DATA_BLOCK "DB_FixReadReal"
{ S7_Optimized_Access := 'FALSE' }
VERSION : 0.0
   STRUCT
      R0 : Real;
      R4 : Real;
      R8 : Real;
      R12 : Real;
      R16 : Real;
      R20 : Real;
      R24 : Real;
      R28 : Real;
      R32 : Real;
      R36 : Real;
      R40 : Real;
      R44 : Real;
      R48 : Real;
      R52 : Real;
      R56 : Real;
      R60 : Real;   // M501.M2 BQ2 actual position mm MLD (zone 1 big wheels part)
      R64 : Real;   // M501.M3 BQ3 actual position mm MLD (zone 2 big wheels part)
      R68 : Real;
      R72 : Real;
      R76 : Real;
      R80 : Real;
      R84 : Real;
      R88 : Real;
      R92 : Real;
      R96 : Real;
      R100 : Real;
      R104 : Real;
      R108 : Real;
      R112 : Real;
      R116 : Real;
      R120 : Real;   // M502.M1 BQ1actual position mm
      R124 : Real;
      R128 : Real;
      R132 : Real;
      R136 : Real;
      R140 : Real;
      R144 : Real;
      R148 : Real;
      R152 : Real;
      R156 : Real;
      R160 : Real;
      R164 : Real;
      R168 : Real;
      R172 : Real;
      R176 : Real;
      R180 : Real;   // M503
      R184 : Real;
      R188 : Real;
      R192 : Real;
      R196 : Real;
      R200 : Real;
      R204 : Real;
      R208 : Real;
      R212 : Real;
      R216 : Real;
      R220 : Real;
      R224 : Real;
      R228 : Real;
      R232 : Real;
      R236 : Real;
      R240 : Real;   // M504
      R244 : Real;
      R248 : Real;
      R252 : Real;
      R256 : Real;
      R260 : Real;
      R264 : Real;
      R268 : Real;
      R272 : Real;
      R276 : Real;
      R280 : Real;
      R284 : Real;
      R288 : Real;
      R292 : Real;
      R296 : Real;
      R300 : Real;   // M505
      R304 : Real;
      R308 : Real;
      R312 : Real;
      R316 : Real;
      R320 : Real;
      R324 : Real;
      R328 : Real;
      R332 : Real;
      R336 : Real;
      R340 : Real;
      R344 : Real;
      R348 : Real;
      R352 : Real;
      R356 : Real;
      R360 : Real;   // M506.M1(left part) BQ1actual position (flow dir.)mm
      R364 : Real;   // M506.M2 (right part) BQ2actual position (flow dir.) mm
      R368 : Real;   // M506 BQ3 (left part lateral) encoder position (mm)
      R372 : Real;   // M506 BQ4 (right part lateral) encoder position (mm)
      R376 : Real;
      R380 : Real;
      R384 : Real;
      R388 : Real;
      R392 : Real;
      R396 : Real;
      R400 : Real;
      R404 : Real;
      R408 : Real;
      R412 : Real;
      R416 : Real;
      R420 : Real;
      R424 : Real;
      R428 : Real;
      R432 : Real;
      R436 : Real;
      R440 : Real;
      R444 : Real;
      R448 : Real;
      R452 : Real;
      R456 : Real;
      R460 : Real;
      R464 : Real;
      R468 : Real;
      R472 : Real;
      R476 : Real;
      R480 : Real;
      R484 : Real;
      R488 : Real;
      R492 : Real;
      R496 : Real;
   END_STRUCT;


BEGIN
   R104 := 6.0;
   R128 := 149.5241;
   R192 := -66.20112;
   R200 := -76.06335;
   R300 := -4029.408;
   R316 := 3331.177;
   R320 := -138.2032;
   R364 := 1.45126E-38;
   R368 := 1984.16;
   R372 := 1140.075;
   R400 := -4.943526;
   R440 := -34.01926;
   R448 := -33.99865;

END_DATA_BLOCK

DATA_BLOCK "DB_FixReadDint"
{ S7_Optimized_Access := 'FALSE' }
VERSION : 0.0
   STRUCT
      DW0 : DInt;   // General.
      DW4 : DInt;
      DW8 : DInt;
      DW12 : DInt;
      DW16 : DInt;
      DW20 : DInt;
      DW24 : DInt;
      DW28 : DInt;
      DW32 : DInt;
      DW36 : DInt;
      DW40 : DInt;
      DW44 : DInt;
      DW48 : DInt;
      DW52 : DInt;
      DW56 : DInt;
      DW60 : DInt;   // M501
      DW64 : DInt;
      DW68 : DInt;
      DW72 : DInt;
      DW76 : DInt;
      DW80 : DInt;
      DW84 : DInt;
      DW88 : DInt;
      DW92 : DInt;
      DW96 : DInt;
      DW100 : DInt;
      DW104 : DInt;
      DW108 : DInt;
      DW112 : DInt;
      DW116 : DInt;
      DW120 : DInt;   // M502
      DW124 : DInt;
      DW128 : DInt;
      DW132 : DInt;
      DW136 : DInt;
      DW140 : DInt;
      DW144 : DInt;
      DW148 : DInt;
      DW152 : DInt;
      DW156 : DInt;
      DW160 : DInt;
      DW164 : DInt;
      DW168 : DInt;
      DW172 : DInt;
      DW176 : DInt;
      DW180 : DInt;   // M503 BQ1 Rotator encoder pulses (reading referenced to starting value)
      DW184 : DInt;
      DW188 : DInt;
      DW192 : DInt;
      DW196 : DInt;
      DW200 : DInt;
      DW204 : DInt;
      DW208 : DInt;
      DW212 : DInt;
      DW216 : DInt;
      DW220 : DInt;
      DW224 : DInt;
      DW228 : DInt;
      DW232 : DInt;
      DW236 : DInt;
      DW240 : DInt;   // M504
      DW244 : DInt;
      DW248 : DInt;
      DW252 : DInt;
      DW256 : DInt;
      DW260 : DInt;
      DW264 : DInt;
      DW268 : DInt;
      DW272 : DInt;
      DW276 : DInt;
      DW280 : DInt;
      DW284 : DInt;
      DW288 : DInt;
      DW292 : DInt;
      DW296 : DInt;
      DW300 : DInt;   // M505
      DW304 : DInt;
      DW308 : DInt;
      DW312 : DInt;
      DW316 : DInt;
      DW320 : DInt;
      DW324 : DInt;
      DW328 : DInt;
      DW332 : DInt;
      DW336 : DInt;
      DW340 : DInt;
      DW344 : DInt;
      DW348 : DInt;
      DW352 : DInt;
      DW356 : DInt;
      DW360 : DInt;   // M506
      DW364 : DInt;   // M506
      DW368 : DInt;   // M506 BQ3 (left part MLD) encoder pulses
      DW372 : DInt;   // M506 BQ4 (right part MLD) encoder pulses
      DW376 : DInt;
      DW380 : DInt;
      DW384 : DInt;
      DW388 : DInt;
      DW392 : DInt;
      DW396 : DInt;
      DW400 : DInt;
      DW404 : DInt;
      DW408 : DInt;
      DW412 : DInt;
      DW416 : DInt;
      DW420 : DInt;
      DW424 : DInt;
      DW428 : DInt;
      DW432 : DInt;
      DW436 : DInt;
      DW440 : DInt;
      DW444 : DInt;
      DW448 : DInt;
      DW452 : DInt;
      DW456 : DInt;
      DW460 : DInt;
      DW464 : DInt;
      DW468 : DInt;
      DW472 : DInt;
      DW476 : DInt;
      DW480 : DInt;   // LES1_M507:BQ1.Encoder position (imp)
      DW484 : DInt;
      DW488 : DInt;
      DW492 : DInt;
      DW496 : DInt;
      DW500 : DInt;
      DW504 : DInt;
      DW508 : DInt;
      DW512 : DInt;
      DW516 : DInt;
      DW520 : DInt;   // LES1_M508:Slide 1.BQ1.Encoder position (imp)
      DW524 : DInt;   // LES1_M508:Slide 2.BQ2.Encoder position (imp)
      DW528 : DInt;   // LES1_M508:Slide 1.BQ1.Encoder position (mm)
      DW532 : DInt;   // LES1_M508:Slide 2.BQ2.Encoder position (mm)
      DW536 : DInt;
      DW540 : DInt;
      DW544 : DInt;
      DW548 : DInt;
      DW552 : DInt;
      DW556 : DInt;
      DW560 : DInt;
      DW564 : DInt;
      DW568 : DInt;
      DW572 : DInt;
      DW576 : DInt;
      DW580 : DInt;
      DW584 : DInt;   // LES1_M508:Rotating platform.BQ3.Encoder position (imp)
      DW588 : DInt;
      DW592 : DInt;
      DW596 : DInt;
      DW600 : DInt;
      DW604 : DInt;
      DW608 : DInt;
      DW612 : DInt;
      DW616 : DInt;
      DW620 : DInt;
      DW624 : DInt;
      DW628 : DInt;
      DW632 : DInt;
      DW636 : DInt;
      DW640 : DInt;
      DW644 : DInt;
      DW648 : DInt;
      DW652 : DInt;
      DW656 : DInt;
      DW660 : DInt;
      DW664 : DInt;
      DW668 : DInt;
      DW672 : DInt;
      DW676 : DInt;
      DW680 : DInt;
      DW684 : DInt;
      DW688 : DInt;
      DW692 : DInt;
      DW696 : DInt;
      DW700 : DInt;
      DW704 : DInt;
      DW708 : DInt;
      DW712 : DInt;
      DW716 : DInt;
      DW720 : DInt;
      DW724 : DInt;
      DW728 : DInt;
      DW732 : DInt;
      DW736 : DInt;
      DW740 : DInt;
      DW744 : DInt;
      DW748 : DInt;
      DW752 : DInt;
      DW756 : DInt;
      DW760 : DInt;
      DW764 : DInt;
      DW768 : DInt;
      DW772 : DInt;
      DW776 : DInt;
      DW780 : DInt;
      DW784 : DInt;
      DW788 : DInt;
      DW792 : DInt;
      DW796 : DInt;
      DW800 : DInt;
      DW804 : DInt;
      DW808 : DInt;
      DW812 : DInt;
      DW816 : DInt;
      DW820 : DInt;
      DW824 : DInt;
      DW828 : DInt;
      DW832 : DInt;
      DW836 : DInt;
      DW840 : DInt;
      DW844 : DInt;
      DW848 : DInt;
      DW852 : DInt;
      DW856 : DInt;
      DW860 : DInt;
      DW864 : DInt;
      DW868 : DInt;
      DW872 : DInt;
      DW876 : DInt;
      DW880 : DInt;
      DW884 : DInt;
      DW888 : DInt;
      DW892 : DInt;
      DW896 : DInt;
   END_STRUCT;


BEGIN
   DW128 := DINT#14373;
   DW368 := DINT#79289;
   DW372 := DINT#27030;
   DW384 := DINT#2300;
   DW392 := DINT#4600;
   DW404 := DINT#3210;
   DW432 := DINT#1605;
   DW480 := DINT#1363;
   DW520 := DINT#7471;
   DW524 := DINT#7728;
   DW528 := DINT#912;
   DW532 := DINT#943;
   DW536 := DINT#91114;
   DW584 := DINT#27181;

END_DATA_BLOCK

DATA_BLOCK "DB_FixReadInt"
{ S7_Optimized_Access := 'FALSE' }
VERSION : 0.0
   STRUCT
      W0 : Int;   // Z500. State zone
      W2 : Int;
      W4 : Int;   // Z500.Mode zone (1=manu  4=auto)
      W6 : Int;
      W8 : Int;
      W10 : Int;   // Z500.selected (1=20;3=40 4=60 5=80 m/min)
      W12 : Int;
      W14 : Int;   // Z500 anomaly on  MCC1501 (1=faute)
      W16 : Int;
      W18 : Int;   // Z500. Line Enable (1=enable 0=no )
      W20 : Int;   // Z500. Line ready to receive glass from Main line (1= ready  0= Not ready)
      W22 : Int;
      W24 : Int;   // Z500.Selection conveyor start clean (M501-M506)(accepted)
      W26 : Int;
      W28 : Int;
      BitNuovi : Struct   // struct created to use this word, relative to "Portrait=1 /Landscape=2" as a bit
         byteMSD : Byte;
         bit0 : Bool;   // Z500.selected Unloading mode =Portrait
         bit1 : Bool;   // Z500.Selected Unloading mode =Landscape
      END_STRUCT;
      W32 : Int;
      W34 : Int;
      W36 : Int;
      W38 : Int;
      W40 : Int;
      W42 : Int;
      W44 : Int;
      W46 : Int;
      W48 : Int;
      W50 : Int;   // M501.M1.Machine state (rollers part)
      W52 : Int;   // M501.M2.Machine state (zone 1 wheels part)
      W54 : Int;   // M501.M3.Machine state (zone 2 wheels part)
      W56 : Int;   // M501.M4.Machine state (glass unload)
      W58 : Int;
      W60 : Int;
      W62 : Int;
      W64 : Int;
      W66 : Int;
      W68 : Int;
      W70 : Int;   // M502.M1.Machine state
      W72 : Int;   // M502_3 Area access status
      W74 : Int;
      W76 : Int;
      W78 : Int;
      W80 : Int;
      W82 : Int;
      W84 : Int;
      W86 : Int;
      W88 : Int;
      W90 : Int;   // M503.Machine state (Rotator device)
      W92 : Int;
      W94 : Int;
      W96 : Int;
      W98 : Int;
      W100 : Int;
      W102 : Int;
      W104 : Int;
      W106 : Int;
      W108 : Int;
      W110 : Int;   // M504.M1 Machine state (left)
      W112 : Int;   // M504.M2 Machine state (right)
      W114 : Int;
      W116 : Int;   // M504 Speed reduction during unpacking status  (0= OFF 1= ON)
      W118 : Int;   // M504 Move Backward enable status (0= OFF 1= ON)
      W120 : Int;
      W122 : Int;
      W124 : Int;
      W126 : Int;
      W128 : Int;
      W130 : Int;   // M505.M1 Machine state (left)
      W132 : Int;   // M505.M2 Machine state (right)
      W134 : Int;
      W136 : Int;
      W138 : Int;
      W140 : Int;
      W142 : Int;
      W144 : Int;
      W146 : Int;
      W148 : Int;
      W150 : Int;   // M506.M1 Machine state (left)
      W152 : Int;   // M506.M2 Machine state (right)
      W154 : Int;   // M506.M3 Machine state (left) MLD
      W156 : Int;   // M506.M4 Machine state (right) MLD
      W158 : Int;   // M506 Right Glass Presence status (1=Loaded 2=Positione 4=Squared) A or Mono
      W160 : Int;   // M506 Left Glass Presence status (1=Loaded 2=Positione 4=Squared) B
      W162 : Int;
      W164 : Int;
      W166 : Int;
      W168 : Int;
      W170 : Int;
      W172 : Int;
      W174 : Int;
      W176 : Int;
      W178 : Int;
      W180 : Int;
      W182 : Int;
      W184 : Int;
      W186 : Int;
      W188 : Int;
      W190 : Int;
      W192 : Int;
      W194 : Int;
      W196 : Int;
      W198 : Int;
      W200 : Int;
      W202 : Int;
      W204 : Int;
      W206 : Int;
      W208 : Int;
      W210 : Int;
      W212 : Int;
      W214 : Int;
      W216 : Int;
      W218 : Int;
      W220 : Int;
      W222 : Int;
      W224 : Int;
      W226 : Int;
      W228 : Int;
      W230 : Int;   // LES1_M507.Entry Zone
      W232 : Int;   // LES1_M507.Entry Zone Barriere Photocell
      W234 : Int;   // LES1_M507.Entry Zone door
      W236 : Int;   // LES1_M507.Cycle Time (s/100)
      W238 : Int;   // LES1_M507.Test Modality (1=Active)
      W240 : Int;   // LES1_M507.Arm Speed selection (1=Selection,0=Thickness)
      W242 : Int;   // LES1_M507 Cups selection in manual(1) or auto(0)
      W244 : Int;
      W246 : Int;
      W248 : Int;
      W250 : Int;
      W252 : Int;
      W254 : Int;
      W256 : Int;
      W258 : Int;
      W260 : Int;   // LES1_M507:State machine(1,3,7)
      W262 : Int;   // LES1_M507:Mode machine(Manu,semiauto,auto) 1,2,4
      W264 : Int;   // LES1_M507.Actual arms speed
      W266 : Int;   // LES1_M507:Status return in line ( 0=NoReentry 1=ReentryReq. 2=ReentryAccepted)
      W268 : Int;
      W270 : Int;   // M507_Z.St.:1=Stop2=Starting3=Run 4=Stop 7=Fault 15=Clean line 16=Emerg. 17=Man
      W272 : Int;
      W274 : Int;
      W276 : Int;   // LES1 :M507 Actual arms position
      W278 : Int;
      W280 : Int;   // LES1_M507:glass presence (0= no glass 1= presence 1 sheet  2=presence 2 sheets)
      W282 : Int;
      W284 : Int;
      W286 : Int;
      W288 : Int;
      W290 : Int;   // LES1_M507.Legth (mm)
      W292 : Int;   // LES1_M507.Whidth (mm)
      W294 : Int;   // LES1_M507.Thickness (mm/100)
      W296 : Int;
      W298 : Int;
      W300 : Int;   // LES1_M507: (0= DISABLED  1= ENABLE)
      W302 : Int;
      W304 : Int;
      W306 : Int;
      W308 : Int;
      W310 : Int;
      W312 : Int;
      W314 : Int;
      W316 : Int;
      W318 : Int;
      W320 : Int;
      W322 : Int;
      W324 : Int;
      W326 : Int;
      W328 : Int;
      W330 : Int;
      W332 : Int;
      W334 : Int;
      W336 : Int;
      W338 : Int;
      W340 : Int;
      W342 : Int;
      W344 : Int;
      W346 : Int;
      W348 : Int;
      W350 : Int;
      W352 : Int;
      W354 : Int;
      W356 : Int;
      W358 : Int;
      W360 : Int;   // LES1_M508:State machine (plateform)
      W362 : Int;   // LES1_M508:State machine (slide 1)
      W364 : Int;   // LES1_M508:State machine (slide 2)
      W366 : Int;   // LES1_M508.Platform Data Source (0=FIX 1=Remote)
      W368 : Int;   // LES1_M508.Platform Rack State 1= aligned side A
      W370 : Int;   // LES1_M508.Platform Rack State 1= aligned side B
      W372 : Int;   // LES1_M508.Platform 0° Side A (0=Not Ready, 1=Ready)
      W374 : Int;   // LES1_M508.Platform 180° Side B (0=Not Ready, 1=Ready)
      W376 : Int;   // LES1_M508.Platform 0°  Set Pack number
      W378 : Int;   // LES1_M508.Platform 0°  Set Sheet number
      W380 : Int;   // LES1_M508.Platform 0° Unloaded Pack
      W382 : Int;   // LES1_M508.Platform 0° Unloaded Sheet
      W384 : Int;
      W386 : Int;   // LES1_M508.Platform 180°  Set Pack number
      W388 : Int;   // LES1_M508.Platform 180°  Set Sheet number
      W390 : Int;   // LES1_M508.Platform 180° Unloaded Pack
      W392 : Int;   // LES1_M508.Platform 180° Unloaded Sheet
      W394 : Int;
      W396 : Int;
      W398 : Int;
      W400 : Int;   // LES1 M508.Slides Selection cycle type (1 = Fixed, 0 = Thickness)
      W402 : Int;
      W404 : Int;
      W406 : Int;
      W408 : Int;
      W410 : Int;
      W412 : Int;
      W414 : Int;
      W416 : Int;
      W418 : Int;
      W420 : Int;
      W422 : Int;
      W424 : Int;
      W426 : Int;
      W428 : Int;
      W430 : Int;   // LES1_M509 left pusher :State machine (1,3,7)
      W432 : Int;   // LES1_M509 right pusher :State machine (1,3,7)
      W434 : Int;
      W436 : Int;
      W438 : Int;
      W440 : Int;
      W442 : Int;
      W444 : Int;
      W446 : Int;
      W448 : Int;
      W450 : Int;
      W452 : Int;
      W454 : Int;
      W456 : Int;
      W458 : Int;
      W460 : Int;
      W462 : Int;
      W464 : Int;
      W466 : Int;
      W468 : Int;
      W470 : Int;
      W472 : Int;
      W474 : Int;
      W476 : Int;
      W478 : Int;
      W480 : Int;
      W482 : Int;
      W484 : Int;
      W486 : Int;
      W488 : Int;
      W490 : Int;
      W492 : Int;
      W494 : Int;
      W496 : Int;
      W498 : Int;
      W500 : Int;
      W502 : Int;
      W504 : Int;
      W506 : Int;
      W508 : Int;
      W510 : Int;
      W512 : Int;
      W514 : Int;
      W516 : Int;
      W518 : Int;
      W520 : Int;
      W522 : Int;
      W524 : Int;
      W526 : Int;
      W528 : Int;
      W530 : Int;
      W532 : Int;
      W534 : Int;
      W536 : Int;
      W538 : Int;
      W540 : Int;
      W542 : Int;
      W544 : Int;
      W546 : Int;
      W548 : Int;
      W550 : Int;
      W552 : Int;
      W554 : Int;
      W556 : Int;
      W558 : Int;
      W560 : Int;
      W562 : Int;
      W564 : Int;
      W566 : Int;
      W568 : Int;
      W570 : Int;
      W572 : Int;
      W574 : Int;
      W576 : Int;
      W578 : Int;
      W580 : Int;
      W582 : Int;
      W584 : Int;
      W586 : Int;
      W588 : Int;
      W590 : Int;
      W592 : Int;
      W594 : Int;
      W596 : Int;
      W598 : Int;
      W600 : Int;
      W602 : Int;
      W604 : Int;
      W606 : Int;
      W608 : Int;
      W610 : Int;
      W612 : Int;
      W614 : Int;
      W616 : Int;
      W618 : Int;
      W620 : Int;
      W622 : Int;
      W624 : Int;
      W626 : Int;
      W628 : Int;
      W630 : Int;
      W632 : Int;
      W634 : Int;
      W636 : Int;
      W638 : Int;
      W640 : Int;
      W642 : Int;
      W644 : Int;
      W646 : Int;
      W648 : Int;
      W650 : Int;
      W652 : Int;
      W654 : Int;
      W656 : Int;
      W658 : Int;
      W660 : Int;
      W662 : Int;
      W664 : Int;
      W666 : Int;
      W668 : Int;
      W670 : Int;
      W672 : Int;
      W674 : Int;
      W676 : Int;
      W678 : Int;
      W680 : Int;
      W682 : Int;
      W684 : Int;
      W686 : Int;
      W688 : Int;
      W690 : Int;
      W692 : Int;
      W694 : Int;
      W696 : Int;
      W698 : Int;
      W700 : Int;
      W702 : Int;
      W704 : Int;
      W706 : Int;
      W708 : Int;
      W710 : Int;
      W712 : Int;
      W714 : Int;
      W716 : Int;
      W718 : Int;
      W720 : Int;
      W722 : Int;
      W724 : Int;
      W726 : Int;
      W728 : Int;
      W730 : Int;
      W732 : Int;
      W734 : Int;
      W736 : Int;
      W738 : Int;
      W740 : Int;
      W742 : Int;
      W744 : Int;
      W746 : Int;
      W748 : Int;
      W750 : Int;
      W752 : Int;
      W754 : Int;
      W756 : Int;
      W758 : Int;
      W760 : Int;
      W762 : Int;
      W764 : Int;
      W766 : Int;
      W768 : Int;
      W770 : Int;
      W772 : Int;
      W774 : Int;
      W776 : Int;
      W778 : Int;
      W780 : Int;
      W782 : Int;
      W784 : Int;
      W786 : Int;
      W788 : Int;
      W790 : Int;
      W792 : Int;
      W794 : Int;
      W796 : Int;
      W798 : Int;
      W800 : Int;
      W802 : Int;
      W804 : Int;
      W806 : Int;
      W808 : Int;
      W810 : Int;
      W812 : Int;
      W814 : Int;
      W816 : Int;
      W818 : Int;
      W820 : Int;
      W822 : Int;
      W824 : Int;
      W826 : Int;
      W828 : Int;
      W830 : Int;
      W832 : Int;
      W834 : Int;
      W836 : Int;
      W838 : Int;
      W840 : Int;
      W842 : Int;
      W844 : Int;
      W846 : Int;
      W848 : Int;
      W850 : Int;
      W852 : Int;
      W854 : Int;
      W856 : Int;
      W858 : Int;
      W860 : Int;
      W862 : Int;
      W864 : Int;
      W866 : Int;
      W868 : Int;
      W870 : Int;
      W872 : Int;
      W874 : Int;
      W876 : Int;
      W878 : Int;
      W880 : Int;
      W882 : Int;
      W884 : Int;
      W886 : Int;
      W888 : Int;
      W890 : Int;
      W892 : Int;
      W894 : Int;
      W896 : Int;
      W898 : Int;
      W900 : Int;
      W902 : Int;
      W904 : Int;
      W906 : Int;
      W908 : Int;
      W910 : Int;
      W912 : Int;
      W914 : Int;
      W916 : Int;
      W918 : Int;
      W920 : Int;
      W922 : Int;
      W924 : Int;
      W926 : Int;
      W928 : Int;
      W930 : Int;
      W932 : Int;
      W934 : Int;
      W936 : Int;
      W938 : Int;
      W940 : Int;
      W942 : Int;
      W944 : Int;
      W946 : Int;
      W948 : Int;
      W950 : Int;
      W952 : Int;
      W954 : Int;
      W956 : Int;
      W958 : Int;
      W960 : Int;
      W962 : Int;
      W964 : Int;
      W966 : Int;
      W968 : Int;
      W970 : Int;
      W972 : Int;
      W974 : Int;
      W976 : Int;
      W978 : Int;
      W980 : Int;
      W982 : Int;
      W984 : Int;
      W986 : Int;
      W988 : Int;
      W990 : Int;
      W992 : Int;
      W994 : Int;
      W996 : Int;
      W998 : Int;
      W1000 : Int;
      W1002 : Int;
      W1004 : Int;
      W1006 : Int;
      W1008 : Int;
      W1010 : Int;
      W1012 : Int;
      W1014 : Int;
      W1016 : Int;
      W1018 : Int;
      W1020 : Int;
      W1022 : Int;
      W1024 : Int;
      W1026 : Int;
      W1028 : Int;
      W1030 : Int;
      W1032 : Int;
      W1034 : Int;
      W1036 : Int;
      W1038 : Int;
      W1040 : Int;
      W1042 : Int;
      W1044 : Int;
      W1046 : Int;
      W1048 : Int;
      W1050 : Int;
      W1052 : Int;
      W1054 : Int;
      W1056 : Int;
      W1058 : Int;
      W1060 : Int;
      W1062 : Int;
      W1064 : Int;
      W1066 : Int;
      W1068 : Int;
      W1070 : Int;
      W1072 : Int;
      W1074 : Int;
      W1076 : Int;
      W1078 : Int;
      W1080 : Int;
      W1082 : Int;
      W1084 : Int;
      W1086 : Int;
      W1088 : Int;
      W1090 : Int;
      W1092 : Int;
      W1094 : Int;
      W1096 : Int;
      W1098 : Int;
      W1100 : Int;
      W1102 : Int;
      W1104 : Int;
      W1106 : Int;
      W1108 : Int;
      W1110 : Int;
      W1112 : Int;
      W1114 : Int;
      W1116 : Int;
      W1118 : Int;
      W1120 : Int;
      W1122 : Int;
      W1124 : Int;
      W1126 : Int;
      W1128 : Int;
      W1130 : Int;
      W1132 : Int;
      W1134 : Int;
      W1136 : Int;
      W1138 : Int;
      W1140 : Int;
      W1142 : Int;
      W1144 : Int;
      W1146 : Int;
      W1148 : Int;
      W1150 : Int;
      W1152 : Int;
      W1154 : Int;
      W1156 : Int;
      W1158 : Int;
      W1160 : Int;
      W1162 : Int;
      W1164 : Int;
      W1166 : Int;
      W1168 : Int;
      W1170 : Int;
      W1172 : Int;
      W1174 : Int;
      W1176 : Int;
      W1178 : Int;
      W1180 : Int;
      W1182 : Int;
      W1184 : Int;
      W1186 : Int;
      W1188 : Int;
      W1190 : Int;
      W1192 : Int;
      W1194 : Int;
      W1196 : Int;
      W1198 : Int;
      W1200 : Int;
      W1202 : Int;
      W1204 : Int;
      W1206 : Int;
      W1208 : Int;
      W1210 : Int;
      W1212 : Int;
      W1214 : Int;
      W1216 : Int;
      W1218 : Int;
      W1220 : Int;
      W1222 : Int;
      W1224 : Int;
      W1226 : Int;
      W1228 : Int;
      W1230 : Int;
      W1232 : Int;
      W1234 : Int;
      W1236 : Int;
      W1238 : Int;
      W1240 : Int;
      W1242 : Int;
      W1244 : Int;
      W1246 : Int;
      W1248 : Int;
      W1250 : Int;
      W1252 : Int;
      W1254 : Int;
      W1256 : Int;
      W1258 : Int;
      W1260 : Int;
      W1262 : Int;
      W1264 : Int;
      W1266 : Int;
      W1268 : Int;
      W1270 : Int;
      W1272 : Int;
      W1274 : Int;
      W1276 : Int;
      W1278 : Int;
      W1280 : Int;
      W1282 : Int;
      W1284 : Int;
      W1286 : Int;
      W1288 : Int;
      W1290 : Int;
      W1292 : Int;
      W1294 : Int;
      W1296 : Int;
      W1298 : Int;
      W1300 : Int;
      W1302 : Int;
      W1304 : Int;
      W1306 : Int;
      W1308 : Int;
      W1310 : Int;
      W1312 : Int;
      W1314 : Int;
      W1316 : Int;
      W1318 : Int;
      W1320 : Int;
      W1322 : Int;
      W1324 : Int;
      W1326 : Int;
      W1328 : Int;
      W1330 : Int;
      W1332 : Int;
      W1334 : Int;
      W1336 : Int;
      W1338 : Int;
      W1340 : Int;
      W1342 : Int;
      W1344 : Int;
      W1346 : Int;
      W1348 : Int;
      W1350 : Int;
      W1352 : Int;
      W1354 : Int;
      W1356 : Int;
      W1358 : Int;
      W1360 : Int;
      W1362 : Int;
      W1364 : Int;
      W1366 : Int;
      W1368 : Int;
      W1370 : Int;
      W1372 : Int;
      W1374 : Int;
      W1376 : Int;
      W1378 : Int;
      W1380 : Int;
      W1382 : Int;
      W1384 : Int;
      W1386 : Int;
      W1388 : Int;
      W1390 : Int;
      W1392 : Int;
      W1394 : Int;
      W1396 : Int;
      W1398 : Int;
      W1400 : Int;
      W1402 : Int;
      W1404 : Int;
      W1406 : Int;
      W1408 : Int;
      W1410 : Int;
      W1412 : Int;
      W1414 : Int;
      W1416 : Int;
      W1418 : Int;
      W1420 : Int;
      W1422 : Int;
      W1424 : Int;
      W1426 : Int;
      W1428 : Int;
      W1430 : Int;
      W1432 : Int;
      W1434 : Int;
      W1436 : Int;
      W1438 : Int;
      W1440 : Int;
      W1442 : Int;
      W1444 : Int;
      W1446 : Int;
      W1448 : Int;
      W1450 : Int;
      W1452 : Int;
      W1454 : Int;
      W1456 : Int;
      W1458 : Int;
      W1460 : Int;
      W1462 : Int;
      W1464 : Int;
      W1466 : Int;
      W1468 : Int;
      W1470 : Int;
      W1472 : Int;
      W1474 : Int;
      W1476 : Int;
      W1478 : Int;
      W1480 : Int;
      W1482 : Int;
      W1484 : Int;
      W1486 : Int;
      W1488 : Int;
      W1490 : Int;
      W1492 : Int;
      W1494 : Int;
      W1496 : Int;
      W1498 : Int;
   END_STRUCT;


BEGIN
   W0 := 3;
   W4 := 4;
   W10 := 4;
   W18 := 1;
   W20 := 1;
   W24 := 506;
   W26 := 505;
   BitNuovi.bit1 := TRUE;
   W50 := 3;
   W52 := 3;
   W54 := 3;
   W56 := 1;
   W60 := 1;
   W62 := 1;
   W64 := 1;
   W66 := 1;
   W68 := 1;
   W70 := 3;
   W74 := 7;
   W76 := 7;
   W78 := 7;
   W80 := 1;
   W82 := 1;
   W84 := 1;
   W86 := 1;
   W90 := 1;
   W92 := 7;
   W100 := 7;
   W110 := 3;
   W112 := 3;
   W118 := 1;
   W130 := 3;
   W132 := 3;
   W146 := 7;
   W150 := 3;
   W152 := 3;
   W154 := 1;
   W156 := 1;
   W166 := 1;
   W170 := 1;
   W172 := 1;
   W174 := 1;
   W178 := 1;
   W190 := 7;
   W192 := 7;
   W210 := 7;
   W218 := 1;
   W220 := 1;
   W230 := 2;
   W232 := 7;
   W234 := 1;
   W240 := 1;
   W250 := 7;
   W252 := 7;
   W258 := 1;
   W260 := 1;
   W262 := 4;
   W264 := 50;
   W270 := 3;
   W276 := 2;
   W278 := 1;
   W290 := 1830;
   W292 := 2440;
   W294 := 500;
   W298 := 1;
   W300 := 2;
   W308 := 1;
   W318 := 1;
   W338 := 1;
   W358 := 1;
   W360 := 7;
   W362 := 7;
   W364 := 1;
   W366 := 1;
   W370 := 1;
   W372 := 1;
   W374 := 1;
   W376 := 1;
   W378 := 45;
   W386 := 1;
   W388 := 45;
   W392 := 4;
   W398 := 7;
   W402 := 16;
   W404 := 3;
   W406 := 1;
   W408 := 1;
   W418 := 7;
   W422 := 7;
   W424 := 75;
   W430 := 1;
   W432 := 1;
   W436 := 6;
   W438 := 7;
   W440 := 1060;
   W442 := 1530;
   W444 := 210;
   W450 := 7;
   W452 := 1;
   W458 := 41;
   W460 := 1;
   W464 := 1;
   W466 := 252;
   W478 := 7;
   W480 := 1;
   W484 := 1;
   W486 := 252;
   W492 := 44;
   W498 := 7;
   W500 := 1;
   W510 := 7;
   W518 := 7;
   W520 := 7;
   W538 := 7;
   W550 := 1;
   W556 := 3;
   W558 := 7;
   W578 := 7;
   W596 := 1;
   W598 := 1;
   W638 := 1;
   W658 := 1;
   W678 := 1;
   W698 := 1;
   W738 := 7;
   W758 := 1;
   W778 := 20;
   W838 := 7;
   W858 := 7;
   W900 := 17;
   W914 := 1;
   W938 := 1;
   W958 := 7;
   W978 := 1;
   W998 := 1;
   W1018 := 1;
   W1038 := 1;
   W1058 := 1;
   W1078 := 1;
   W1098 := 1;
   W1118 := 7;
   W1138 := 7;
   W1158 := 7;
   W1236 := 1;
   W1238 := 1;
   W1240 := 1;
   W1242 := 1;
   W1276 := 1;
   W1278 := 1;
   W1280 := 1;
   W1282 := 1;
   W1320 := 17;
   W1322 := 1;
   W1324 := 3;
   W1358 := 7;
   W1398 := 7;

END_DATA_BLOCK

DATA_BLOCK "DB_FixReadBit"
{ S7_Optimized_Access := 'FALSE' }
VERSION : 0.0
   STRUCT
      b00 : Bool;   // A 32.0 oZ500-MCC1302-Lateral line enabled
      b01 : Bool;   // A 32.1 oZ500-MCC1302- Ready for Cap of lengh <=1830 mm
      b02 : Bool;   // A 32.2 oZ500-MCC1302-Ready for Cap of length > 1830 mm
      b03 : Bool;   // A 32.3 oZ500-MCC1302-Glass clearing lamp for M319
      b04 : Bool;   // A 32.4 oZ500-MCC1302-Unloading >> M319 in progress
      b05 : Bool;
      b06 : Bool;
      b07 : Bool;
      b10 : Bool;   // E      18.0 iZ500-MCC1302-Syncronisation by line -cap arriving
      b11 : Bool;   // E      18.1 iZ500-MCC1302-No convoy request by line
      b12 : Bool;   // E      18.2 iZ500-MCC1302-Speed by line bit 0
      b13 : Bool;   // E      18.3 iZ500-MCC1302-Speed by line bit 1
      b14 : Bool;   // E      18.4 iZ500-MCC1302-glass on tilting machine < in length of "2000 mm"
      b15 : Bool;   // E      18.5 iZ500-MCC1302-glass call clearing p.b.:M319SB4
      b16 : Bool;   // E      18.6 iZ500-MCC1302-Request disable consents by arriving SQC plate
      b17 : Bool;
      b20 : Bool;
      b21 : Bool;
      b22 : Bool;   // Z500.Force mono mode (0=not actived 1=actived)
      b23 : Bool;
      b24 : Bool;
      b25 : Bool;
      b26 : Bool;
      b27 : Bool;
      b30 : Bool;
      b31 : Bool;
      b32 : Bool;
      b33 : Bool;
      b34 : Bool;
      b35 : Bool;
      b36 : Bool;
      b37 : Bool;
      b40 : Bool;   // M501. P142KA1 photocell for positioning on M2/M3  (Start count)E67.2
      b41 : Bool;   // M501-B2 photocell of glass stop for SQC E4.0
      b42 : Bool;   // M501-B3 photocell of unpacking right side E4.1 (not really present)
      b43 : Bool;   // M501-B4 photocell of unpacking left side E4.2 (not really present)
      b44 : Bool;
      b45 : Bool;
      b46 : Bool;
      b47 : Bool;
      b50 : Bool;   // M501.P145KA1small wheels frame to high position E67.7
      b51 : Bool;
      b52 : Bool;
      b53 : Bool;
      b54 : Bool;
      b55 : Bool;
      b56 : Bool;
      b57 : Bool;
      b60 : Bool;   // M502-B1-B2 P146KA1 photocell for positioning during load E68.3
      b61 : Bool;
      b62 : Bool;
      b63 : Bool;
      b64 : Bool;
      b65 : Bool;
      b66 : Bool;
      b67 : Bool;
      b70 : Bool;
      b71 : Bool;
      b72 : Bool;
      b73 : Bool;
      b74 : Bool;
      b75 : Bool;
      b76 : Bool;
      b77 : Bool;
      b80 : Bool;   // M503 P148KA1 Frame to high position E69.0
      b81 : Bool;   // M503 P148KA2 Frame to low position E69.1
      b82 : Bool;   // M503-SQ1 Centering device confirm position E4.3
      b83 : Bool;   // M503-SQ4 Centering device opened (rot.allowed)E4.4
      b84 : Bool;   // M503-SQ5 Centering device closed (rot.not allowed)E4.5
      b85 : Bool;
      b86 : Bool;
      b87 : Bool;   // M503 request of rotation (1= request of rotation 0= no request of rotation)
      b90 : Bool;   // M503 glass rotated (1= rotated 0= not rotated)
      b91 : Bool;
      b92 : Bool;
      b93 : Bool;   // M502-M503 (area saferies)
      b94 : Bool;
      b95 : Bool;
      b96 : Bool;
      b97 : Bool;
      b100 : Bool;   // M504-B1 Glass sheet stop left transport E5.6
      b101 : Bool;   // M504-B2 Glass sheet stop right transport E5.7
      b102 : Bool;   // M504-B3 Glass sheet syncronisation left transport E7.4
      b103 : Bool;   // M504-B4 Glass sheet syncronisation right transport E7.5
      b104 : Bool;
      b105 : Bool;
      b106 : Bool;
      b107 : Bool;
      b110 : Bool;
      b111 : Bool;
      b112 : Bool;
      b113 : Bool;
      b114 : Bool;
      b115 : Bool;
      b116 : Bool;
      b117 : Bool;
      b120 : Bool;   // M505-B3 P173KA1 Glass sheet stop left E75.4
      b121 : Bool;   // M505-B4 P174KA1 Glass sheet stop right E75.6
      b122 : Bool;   // M505-B1 Glass sheet slowdown left transport E6.7
      b123 : Bool;   // M505-B2 Glass sheet slowdown right transport E7.0
      b124 : Bool;
      b125 : Bool;   // M505-SQ4 Frontal squaring upper position E7.2
      b126 : Bool;
      b127 : Bool;
      b130 : Bool;
      b131 : Bool;
      b132 : Bool;
      b133 : Bool;
      b134 : Bool;
      b135 : Bool;
      b136 : Bool;
      b137 : Bool;
      b140 : Bool;   // M506-B11 Glass sheet stop left E7.6
      b141 : Bool;   // M506-SQ11 stop backward translation left photocell E7.7
      b142 : Bool;   // M506-SQ12 stop forward translation left photocell E8.0
      b143 : Bool;   // M506-B21 Glass sheet stop right E8.1
      b144 : Bool;   // M506-SQ21 stop backward translation right photocell E8.2
      b145 : Bool;   // M506-SQ22 stop forward translation right photocell E8.3
      b146 : Bool;   // M506 -P177KA1 Frame to high position E76.4
      b147 : Bool;
      b150 : Bool;
      b151 : Bool;
      b152 : Bool;
      b153 : Bool;
      b154 : Bool;
      b155 : Bool;
      b156 : Bool;
      b157 : Bool;
      b160 : Bool;   // LES1_M507.Indexing (B1 E8.7)
      b161 : Bool;   // LES1_M507.Compressed air pressure (SP1 E9.4)
      b162 : Bool;   // LES1_M507.Change inclination backward (SQ1 E9.7)
      b163 : Bool;   // LES1_M507.Change inclination to middle (SQ2 E9.2)
      b164 : Bool;   // LES1_M507.Change inclination forward (SQ3 E9.3)
      b165 : Bool;   // LES1_M507.Preindexing (B2 E9.0)
      b166 : Bool;   // LES1_M507.Vacuum presence (SP3 E9.3)
      b167 : Bool;   // LES1_M507.Indexing do deposit (SQ4 E10.0)
      b170 : Bool;   // LES1_M507.Indexing to index (SQ5 E10.1)
      b171 : Bool;
      b172 : Bool;
      b173 : Bool;
      b174 : Bool;
      b175 : Bool;
      b176 : Bool;
      b177 : Bool;
      b180 : Bool;   // LES1_M507.Enabled cups groupe "A/E"
      b181 : Bool;   // LES1_M507.Enabled cups groupe "B/E"
      b182 : Bool;   // LES1_M507.Enabled cups groupe "C/E"
      b183 : Bool;   // LES1_M507.Enabled cups groupe "D/E"
      b184 : Bool;
      b185 : Bool;   // LES1_M507.Enabled cups groupe "B/F"
      b186 : Bool;   // LES1_M507.Enabled cups groupe "C/F"
      b187 : Bool;   // LES1_M507.Enabled cups groupe "D/F"
      b190 : Bool;   // LES1_M507.Enabled cups groupe "A/G"
      b191 : Bool;   // LES1_M507.Enabled cups groupe "B/G"
      b192 : Bool;   // LES1_M507.Enabled cups groupe "C/G"
      b193 : Bool;   // LES1_M507.Enabled cups groupe "D/G"
      b194 : Bool;
      b195 : Bool;
      b196 : Bool;
      b197 : Bool;
      b200 : Bool;
      b201 : Bool;
      b202 : Bool;
      b203 : Bool;
      b204 : Bool;
      b205 : Bool;
      b206 : Bool;
      b207 : Bool;
      b210 : Bool;
      b211 : Bool;
      b212 : Bool;
      b213 : Bool;
      b214 : Bool;
      b215 : Bool;
      b216 : Bool;
      b217 : Bool;
      b220 : Bool;   // LES1_M508.Stop forward carriage 1
      b221 : Bool;   // LES1_M508.Stop backward carriage 1
      b222 : Bool;   // LES1_M508.Stop forward carriage 2
      b223 : Bool;   // LES1_M508.Stop backward carriage 2
      b224 : Bool;   // LES1_M508.Centering device open
      b225 : Bool;
      b226 : Bool;
      b227 : Bool;
      b230 : Bool;   // LES1_M508.Platform 0° Position [Side A]
      b231 : Bool;   // LES1_M508.Platform 180° Position [Side B]
      b232 : Bool;
      b233 : Bool;
      b234 : Bool;
      b235 : Bool;
      b236 : Bool;
      b237 : Bool;   // LES1_M508.Platform.End Pack 0° [Side A]
      b240 : Bool;   // LES1_M508.Platform.End Pack 0° [Side A]
      b241 : Bool;   // LES1_M508.Platform.End Pack 180° [Side B]
      b242 : Bool;   // LES1_M508.Platform.End Rack 0° [Side A]
      b243 : Bool;   // LES1_M508.Platform.End Rack 180° [Side B]
      b244 : Bool;   // LES1_M508.Platform.Rack Ready side A (not used by Fix)
      b245 : Bool;   // LES1_M508.Platform.Rack Ready side B  (not used by Fix)
      b246 : Bool;
      b247 : Bool;
      b250 : Bool;
      b251 : Bool;
      b252 : Bool;
      b253 : Bool;
      b254 : Bool;
      b255 : Bool;
      b256 : Bool;
      b257 : Bool;
      b260 : Bool;   // LES1_M509. Right Pushers enabled
      b261 : Bool;   // LES1_M509. Left  Pusher enabled
      b262 : Bool;
      b263 : Bool;
      b264 : Bool;
      b265 : Bool;
      b266 : Bool;
      b267 : Bool;
      b270 : Bool;
      b271 : Bool;
      b272 : Bool;
      b273 : Bool;
      b274 : Bool;
      b275 : Bool;
      b276 : Bool;
      b277 : Bool;
      b280 : Bool;
      b281 : Bool;
      b282 : Bool;
      b283 : Bool;
      b284 : Bool;
      b285 : Bool;
      b286 : Bool;
      b287 : Bool;
      b290 : Bool;
      b291 : Bool;
      b292 : Bool;
      b293 : Bool;
      b294 : Bool;
      b295 : Bool;
      b296 : Bool;
      b297 : Bool;
      b300 : Bool;
      b301 : Bool;
      b302 : Bool;
      b303 : Bool;
      b304 : Bool;
      b305 : Bool;
      b306 : Bool;
      b307 : Bool;
      b310 : Bool;
      b311 : Bool;
      b312 : Bool;
      b313 : Bool;
      b314 : Bool;
      b315 : Bool;
      b316 : Bool;
      b317 : Bool;
      b320 : Bool;
      b321 : Bool;
      b322 : Bool;
      b323 : Bool;
      b324 : Bool;
      b325 : Bool;
      b326 : Bool;
      b327 : Bool;
      b330 : Bool;
      b331 : Bool;
      b332 : Bool;
      b333 : Bool;
      b334 : Bool;
      b335 : Bool;
      b336 : Bool;
      b337 : Bool;
      b340 : Bool;
      b341 : Bool;
      b342 : Bool;
      b343 : Bool;
      b344 : Bool;
      b345 : Bool;
      b346 : Bool;
      b347 : Bool;
      b350 : Bool;
      b351 : Bool;
      b352 : Bool;
      b353 : Bool;
      b354 : Bool;
      b355 : Bool;
      b356 : Bool;
      b357 : Bool;
      b360 : Bool;
      b361 : Bool;
      b362 : Bool;
      b363 : Bool;
      b364 : Bool;
      b365 : Bool;
      b366 : Bool;
      b367 : Bool;
      b370 : Bool;
      b371 : Bool;
      b372 : Bool;
      b373 : Bool;
      b374 : Bool;
      b375 : Bool;
      b376 : Bool;
      b377 : Bool;
      b380 : Bool;
      b381 : Bool;
      b382 : Bool;
      b383 : Bool;
      b384 : Bool;
      b385 : Bool;
      b386 : Bool;
      b387 : Bool;
      b390 : Bool;
      b391 : Bool;
      b392 : Bool;
      b393 : Bool;
      b394 : Bool;
      b395 : Bool;
      b396 : Bool;
      b397 : Bool;
      b400 : Bool;
      b401 : Bool;
      b402 : Bool;
      b403 : Bool;
      b404 : Bool;
      b405 : Bool;
      b406 : Bool;
      b407 : Bool;
      b410 : Bool;
      b411 : Bool;
      b412 : Bool;
      b413 : Bool;
      b414 : Bool;
      b415 : Bool;
      b416 : Bool;
      b417 : Bool;
      b420 : Bool;
      b421 : Bool;
      b422 : Bool;
      b423 : Bool;
      b424 : Bool;
      b425 : Bool;
      b426 : Bool;
      b427 : Bool;
      b430 : Bool;
      b431 : Bool;
      b432 : Bool;
      b433 : Bool;
      b434 : Bool;
      b435 : Bool;
      b436 : Bool;
      b437 : Bool;
      b440 : Bool;
      b441 : Bool;
      b442 : Bool;
      b443 : Bool;
      b444 : Bool;
      b445 : Bool;
      b446 : Bool;
      b447 : Bool;
      b450 : Bool;
      b451 : Bool;
      b452 : Bool;
      b453 : Bool;
      b454 : Bool;
      b455 : Bool;
      b456 : Bool;
      b457 : Bool;
      b460 : Bool;
      b461 : Bool;
      b462 : Bool;
      b463 : Bool;
      b464 : Bool;
      b465 : Bool;
      b466 : Bool;
      b467 : Bool;
      b470 : Bool;
      b471 : Bool;
      b472 : Bool;
      b473 : Bool;
      b474 : Bool;
      b475 : Bool;
      b476 : Bool;
      b477 : Bool;
      b480 : Bool;
      b481 : Bool;
      b482 : Bool;
      b483 : Bool;
      b484 : Bool;
      b485 : Bool;
      b486 : Bool;
      b487 : Bool;
      b490 : Bool;
      b491 : Bool;
      b492 : Bool;
      b493 : Bool;
      b494 : Bool;
      b495 : Bool;
      b496 : Bool;
      b497 : Bool;
      b500 : Bool;
      b501 : Bool;
      b502 : Bool;
      b503 : Bool;
      b504 : Bool;
      b505 : Bool;
      b506 : Bool;
      b507 : Bool;
      b510 : Bool;
      b511 : Bool;
      b512 : Bool;
      b513 : Bool;
      b514 : Bool;
      b515 : Bool;
      b516 : Bool;
      b517 : Bool;
      b520 : Bool;
      b521 : Bool;
      b522 : Bool;
      b523 : Bool;
      b524 : Bool;
      b525 : Bool;
      b526 : Bool;
      b527 : Bool;
      b530 : Bool;
      b531 : Bool;
      b532 : Bool;
      b533 : Bool;
      b534 : Bool;
      b535 : Bool;
      b536 : Bool;
      b537 : Bool;
      b540 : Bool;
      b541 : Bool;
      b542 : Bool;
      b543 : Bool;
      b544 : Bool;
      b545 : Bool;
      b546 : Bool;
      b547 : Bool;
      b550 : Bool;
      b551 : Bool;
      b552 : Bool;
      b553 : Bool;
      b554 : Bool;
      b555 : Bool;
      b556 : Bool;
      b557 : Bool;
      b560 : Bool;
      b561 : Bool;
      b562 : Bool;
      b563 : Bool;
      b564 : Bool;
      b565 : Bool;
      b566 : Bool;
      b567 : Bool;
      b570 : Bool;
      b571 : Bool;
      b572 : Bool;
      b573 : Bool;
      b574 : Bool;
      b575 : Bool;
      b576 : Bool;
      b577 : Bool;
      b580 : Bool;
      b581 : Bool;
      b582 : Bool;
      b583 : Bool;
      b584 : Bool;
      b585 : Bool;
      b586 : Bool;
      b587 : Bool;
      b590 : Bool;
      b591 : Bool;
      b592 : Bool;
      b593 : Bool;
      b594 : Bool;
      b595 : Bool;
      b596 : Bool;
      b597 : Bool;
      b600 : Bool;
      b601 : Bool;
      b602 : Bool;
      b603 : Bool;
      b604 : Bool;
      b605 : Bool;
      b606 : Bool;
      b607 : Bool;
      b610 : Bool;
      b611 : Bool;
      b612 : Bool;
      b613 : Bool;
      b614 : Bool;
      b615 : Bool;
      b616 : Bool;
      b617 : Bool;
      b620 : Bool;
      b621 : Bool;
      b622 : Bool;
      b623 : Bool;
      b624 : Bool;
      b625 : Bool;
      b626 : Bool;
      b627 : Bool;
      b630 : Bool;
      b631 : Bool;
      b632 : Bool;
      b633 : Bool;
      b634 : Bool;
      b635 : Bool;
      b636 : Bool;
      b637 : Bool;
      b640 : Bool;
      b641 : Bool;
      b642 : Bool;
      b643 : Bool;
      b644 : Bool;
      b645 : Bool;
      b646 : Bool;
      b647 : Bool;
      b650 : Bool;
      b651 : Bool;
      b652 : Bool;
      b653 : Bool;
      b654 : Bool;
      b655 : Bool;
      b656 : Bool;
      b657 : Bool;
      b660 : Bool;
      b661 : Bool;
      b662 : Bool;
      b663 : Bool;
      b664 : Bool;
      b665 : Bool;
      b666 : Bool;
      b667 : Bool;
      b670 : Bool;
      b671 : Bool;
      b672 : Bool;
      b673 : Bool;
      b674 : Bool;
      b675 : Bool;
      b676 : Bool;
      b677 : Bool;
      b680 : Bool;
      b681 : Bool;
      b682 : Bool;
      b683 : Bool;
      b684 : Bool;
      b685 : Bool;
      b686 : Bool;
      b687 : Bool;
      b690 : Bool;
      b691 : Bool;
      b692 : Bool;
      b693 : Bool;
      b694 : Bool;
      b695 : Bool;
      b696 : Bool;
      b697 : Bool;
      b700 : Bool;
      b701 : Bool;
      b702 : Bool;
      b703 : Bool;
      b704 : Bool;
      b705 : Bool;
      b706 : Bool;
      b707 : Bool;
      b710 : Bool;
      b711 : Bool;
      b712 : Bool;
      b713 : Bool;
      b714 : Bool;
      b715 : Bool;
      b716 : Bool;
      b717 : Bool;
      b720 : Bool;
      b721 : Bool;
      b722 : Bool;
      b723 : Bool;
      b724 : Bool;
      b725 : Bool;
      b726 : Bool;
      b727 : Bool;
      b730 : Bool;
      b731 : Bool;
      b732 : Bool;
      b733 : Bool;
      b734 : Bool;
      b735 : Bool;
      b736 : Bool;
      b737 : Bool;
      b740 : Bool;
      b741 : Bool;
      b742 : Bool;
      b743 : Bool;
      b744 : Bool;
      b745 : Bool;
      b746 : Bool;
      b747 : Bool;
      b750 : Bool;
      b751 : Bool;
      b752 : Bool;
      b753 : Bool;
      b754 : Bool;
      b755 : Bool;
      b756 : Bool;
      b757 : Bool;
      b760 : Bool;
      b761 : Bool;
      b762 : Bool;
      b763 : Bool;
      b764 : Bool;
      b765 : Bool;
      b766 : Bool;
      b767 : Bool;
      b770 : Bool;
      b771 : Bool;
      b772 : Bool;
      b773 : Bool;
      b774 : Bool;
      b775 : Bool;
      b776 : Bool;
      b777 : Bool;
      b780 : Bool;
      b781 : Bool;
      b782 : Bool;
      b783 : Bool;
      b784 : Bool;
      b785 : Bool;
      b786 : Bool;
      b787 : Bool;
      b790 : Bool;
      b791 : Bool;
      b792 : Bool;
      b793 : Bool;
      b794 : Bool;
      b795 : Bool;
      b796 : Bool;
      b797 : Bool;
      b800 : Bool;
      b801 : Bool;
      b802 : Bool;
      b803 : Bool;
      b804 : Bool;
      b805 : Bool;
      b806 : Bool;
      b807 : Bool;
      b810 : Bool;
      b811 : Bool;
      b812 : Bool;
      b813 : Bool;
      b814 : Bool;
      b815 : Bool;
      b816 : Bool;
      b817 : Bool;
      b820 : Bool;
      b821 : Bool;
      b822 : Bool;
      b823 : Bool;
      b824 : Bool;
      b825 : Bool;
      b826 : Bool;
      b827 : Bool;
      b830 : Bool;
      b831 : Bool;
      b832 : Bool;
      b833 : Bool;
      b834 : Bool;
      b835 : Bool;
      b836 : Bool;
      b837 : Bool;
      b840 : Bool;
      b841 : Bool;
      b842 : Bool;
      b843 : Bool;
      b844 : Bool;
      b845 : Bool;
      b846 : Bool;
      b847 : Bool;
      b850 : Bool;
      b851 : Bool;
      b852 : Bool;
      b853 : Bool;
      b854 : Bool;
      b855 : Bool;
      b856 : Bool;
      b857 : Bool;
      b860 : Bool;
      b861 : Bool;
      b862 : Bool;
      b863 : Bool;
      b864 : Bool;
      b865 : Bool;
      b866 : Bool;
      b867 : Bool;
      b870 : Bool;
      b871 : Bool;
      b872 : Bool;
      b873 : Bool;
      b874 : Bool;
      b875 : Bool;
      b876 : Bool;
      b877 : Bool;
      b880 : Bool;
      b881 : Bool;
      b882 : Bool;
      b883 : Bool;
      b884 : Bool;
      b885 : Bool;
      b886 : Bool;
      b887 : Bool;
      b890 : Bool;
      b891 : Bool;
      b892 : Bool;
      b893 : Bool;
      b894 : Bool;
      b895 : Bool;
      b896 : Bool;
      b897 : Bool;
      b900 : Bool;
      b901 : Bool;
      b902 : Bool;
      b903 : Bool;
      b904 : Bool;
      b905 : Bool;
      b906 : Bool;
      b907 : Bool;
      b910 : Bool;
      b911 : Bool;
      b912 : Bool;
      b913 : Bool;
      b914 : Bool;
      b915 : Bool;
      b916 : Bool;
      b917 : Bool;
      b920 : Bool;
      b921 : Bool;
      b922 : Bool;
      b923 : Bool;
      b924 : Bool;
      b925 : Bool;
      b926 : Bool;
      b927 : Bool;
      b930 : Bool;
      b931 : Bool;
      b932 : Bool;
      b933 : Bool;
      b934 : Bool;
      b935 : Bool;
      b936 : Bool;
      b937 : Bool;
      b940 : Bool;
      b941 : Bool;
      b942 : Bool;
      b943 : Bool;
      b944 : Bool;
      b945 : Bool;
      b946 : Bool;
      b947 : Bool;
      b950 : Bool;
      b951 : Bool;
      b952 : Bool;
      b953 : Bool;
      b954 : Bool;
      b955 : Bool;
      b956 : Bool;
      b957 : Bool;
      b960 : Bool;
      b961 : Bool;
      b962 : Bool;
      b963 : Bool;
      b964 : Bool;
      b965 : Bool;
      b966 : Bool;
      b967 : Bool;
      b970 : Bool;
      b971 : Bool;
      b972 : Bool;
      b973 : Bool;
      b974 : Bool;
      b975 : Bool;
      b976 : Bool;
      b977 : Bool;
      b980 : Bool;
      b981 : Bool;
      b982 : Bool;
      b983 : Bool;
      b984 : Bool;
      b985 : Bool;
      b986 : Bool;
      b987 : Bool;
      b990 : Bool;
      b991 : Bool;
      b992 : Bool;
      b993 : Bool;
      b994 : Bool;
      b995 : Bool;
      b996 : Bool;
      b997 : Bool;
      b1000 : Bool;
      b1001 : Bool;
      b1002 : Bool;
      b1003 : Bool;
      b1004 : Bool;
      b1005 : Bool;
      b1006 : Bool;
      b1007 : Bool;
      b1010 : Bool;
      b1011 : Bool;
      b1012 : Bool;
      b1013 : Bool;
      b1014 : Bool;
      b1015 : Bool;
      b1016 : Bool;
      b1017 : Bool;
      b1020 : Bool;
      b1021 : Bool;
      b1022 : Bool;
      b1023 : Bool;
      b1024 : Bool;
      b1025 : Bool;
      b1026 : Bool;
      b1027 : Bool;
      b1030 : Bool;
      b1031 : Bool;
      b1032 : Bool;
      b1033 : Bool;
      b1034 : Bool;
      b1035 : Bool;
      b1036 : Bool;
      b1037 : Bool;
      b1040 : Bool;
      b1041 : Bool;
      b1042 : Bool;
      b1043 : Bool;
      b1044 : Bool;
      b1045 : Bool;
      b1046 : Bool;
      b1047 : Bool;
      b1050 : Bool;
      b1051 : Bool;
      b1052 : Bool;
      b1053 : Bool;
      b1054 : Bool;
      b1055 : Bool;
      b1056 : Bool;
      b1057 : Bool;
      b1060 : Bool;
      b1061 : Bool;
      b1062 : Bool;
      b1063 : Bool;
      b1064 : Bool;
      b1065 : Bool;
      b1066 : Bool;
      b1067 : Bool;
      b1070 : Bool;
      b1071 : Bool;
      b1072 : Bool;
      b1073 : Bool;
      b1074 : Bool;
      b1075 : Bool;
      b1076 : Bool;
      b1077 : Bool;
      b1080 : Bool;
      b1081 : Bool;
      b1082 : Bool;
      b1083 : Bool;
      b1084 : Bool;
      b1085 : Bool;
      b1086 : Bool;
      b1087 : Bool;
      b1090 : Bool;
      b1091 : Bool;
      b1092 : Bool;
      b1093 : Bool;
      b1094 : Bool;
      b1095 : Bool;
      b1096 : Bool;
      b1097 : Bool;
      b1100 : Bool;
      b1101 : Bool;
      b1102 : Bool;
      b1103 : Bool;
      b1104 : Bool;
      b1105 : Bool;
      b1106 : Bool;
      b1107 : Bool;
      b1110 : Bool;
      b1111 : Bool;
      b1112 : Bool;
      b1113 : Bool;
      b1114 : Bool;
      b1115 : Bool;
      b1116 : Bool;
      b1117 : Bool;
      b1120 : Bool;
      b1121 : Bool;
      b1122 : Bool;
      b1123 : Bool;
      b1124 : Bool;
      b1125 : Bool;
      b1126 : Bool;
      b1127 : Bool;
      b1130 : Bool;
      b1131 : Bool;
      b1132 : Bool;
      b1133 : Bool;
      b1134 : Bool;
      b1135 : Bool;
      b1136 : Bool;
      b1137 : Bool;
      b1140 : Bool;
      b1141 : Bool;
      b1142 : Bool;
      b1143 : Bool;
      b1144 : Bool;
      b1145 : Bool;
      b1146 : Bool;
      b1147 : Bool;
      b1150 : Bool;
      b1151 : Bool;
      b1152 : Bool;
      b1153 : Bool;
      b1154 : Bool;
      b1155 : Bool;
      b1156 : Bool;
      b1157 : Bool;
      b1160 : Bool;
      b1161 : Bool;
      b1162 : Bool;
      b1163 : Bool;
      b1164 : Bool;
      b1165 : Bool;
      b1166 : Bool;
      b1167 : Bool;
      b1170 : Bool;
      b1171 : Bool;
      b1172 : Bool;
      b1173 : Bool;
      b1174 : Bool;
      b1175 : Bool;
      b1176 : Bool;
      b1177 : Bool;
      b1180 : Bool;
      b1181 : Bool;
      b1182 : Bool;
      b1183 : Bool;
      b1184 : Bool;
      b1185 : Bool;
      b1186 : Bool;
      b1187 : Bool;
      b1190 : Bool;
      b1191 : Bool;
      b1192 : Bool;
      b1193 : Bool;
      b1194 : Bool;
      b1195 : Bool;
      b1196 : Bool;
      b1197 : Bool;
      b1200 : Bool;
      b1201 : Bool;
      b1202 : Bool;
      b1203 : Bool;
      b1204 : Bool;
      b1205 : Bool;
      b1206 : Bool;
      b1207 : Bool;
      b1210 : Bool;
      b1211 : Bool;
      b1212 : Bool;
      b1213 : Bool;
      b1214 : Bool;
      b1215 : Bool;
      b1216 : Bool;
      b1217 : Bool;
      b1220 : Bool;
      b1221 : Bool;
      b1222 : Bool;
      b1223 : Bool;
      b1224 : Bool;
      b1225 : Bool;
      b1226 : Bool;
      b1227 : Bool;
      b1230 : Bool;
      b1231 : Bool;
      b1232 : Bool;
      b1233 : Bool;
      b1234 : Bool;
      b1235 : Bool;
      b1236 : Bool;
      b1237 : Bool;
      b1240 : Bool;
      b1241 : Bool;
      b1242 : Bool;
      b1243 : Bool;
      b1244 : Bool;
      b1245 : Bool;
      b1246 : Bool;
      b1247 : Bool;
      b1250 : Bool;
      b1251 : Bool;
      b1252 : Bool;
      b1253 : Bool;
      b1254 : Bool;
      b1255 : Bool;
      b1256 : Bool;
      b1257 : Bool;
      b1260 : Bool;
      b1261 : Bool;
      b1262 : Bool;
      b1263 : Bool;
      b1264 : Bool;
      b1265 : Bool;
      b1266 : Bool;
      b1267 : Bool;
      b1270 : Bool;
      b1271 : Bool;
      b1272 : Bool;
      b1273 : Bool;
      b1274 : Bool;
      b1275 : Bool;
      b1276 : Bool;
      b1277 : Bool;
      b1280 : Bool;
      b1281 : Bool;
      b1282 : Bool;
      b1283 : Bool;
      b1284 : Bool;
      b1285 : Bool;
      b1286 : Bool;
      b1287 : Bool;
      b1290 : Bool;
      b1291 : Bool;
      b1292 : Bool;
      b1293 : Bool;
      b1294 : Bool;
      b1295 : Bool;
      b1296 : Bool;
      b1297 : Bool;
      b1300 : Bool;
      b1301 : Bool;
      b1302 : Bool;
      b1303 : Bool;
      b1304 : Bool;
      b1305 : Bool;
      b1306 : Bool;
      b1307 : Bool;
      b1310 : Bool;
      b1311 : Bool;
      b1312 : Bool;
      b1313 : Bool;
      b1314 : Bool;
      b1315 : Bool;
      b1316 : Bool;
      b1317 : Bool;
      b1320 : Bool;
      b1321 : Bool;
      b1322 : Bool;
      b1323 : Bool;
      b1324 : Bool;
      b1325 : Bool;
      b1326 : Bool;
      b1327 : Bool;
      b1330 : Bool;
      b1331 : Bool;
      b1332 : Bool;
      b1333 : Bool;
      b1334 : Bool;
      b1335 : Bool;
      b1336 : Bool;
      b1337 : Bool;
      b1340 : Bool;
      b1341 : Bool;
      b1342 : Bool;
      b1343 : Bool;
      b1344 : Bool;
      b1345 : Bool;
      b1346 : Bool;
      b1347 : Bool;
      b1350 : Bool;
      b1351 : Bool;
      b1352 : Bool;
      b1353 : Bool;
      b1354 : Bool;
      b1355 : Bool;
      b1356 : Bool;
      b1357 : Bool;
      b1360 : Bool;
      b1361 : Bool;
      b1362 : Bool;
      b1363 : Bool;
      b1364 : Bool;
      b1365 : Bool;
      b1366 : Bool;
      b1367 : Bool;
      b1370 : Bool;
      b1371 : Bool;
      b1372 : Bool;
      b1373 : Bool;
      b1374 : Bool;
      b1375 : Bool;
      b1376 : Bool;
      b1377 : Bool;
      b1380 : Bool;
      b1381 : Bool;
      b1382 : Bool;
      b1383 : Bool;
      b1384 : Bool;
      b1385 : Bool;
      b1386 : Bool;
      b1387 : Bool;
      b1390 : Bool;
      b1391 : Bool;
      b1392 : Bool;
      b1393 : Bool;
      b1394 : Bool;
      b1395 : Bool;
      b1396 : Bool;
      b1397 : Bool;
      b1400 : Bool;
      b1401 : Bool;
      b1402 : Bool;
      b1403 : Bool;
      b1404 : Bool;
      b1405 : Bool;
      b1406 : Bool;
      b1407 : Bool;
      b1410 : Bool;
      b1411 : Bool;
      b1412 : Bool;
      b1413 : Bool;
      b1414 : Bool;
      b1415 : Bool;
      b1416 : Bool;
      b1417 : Bool;
      b1420 : Bool;
      b1421 : Bool;
      b1422 : Bool;
      b1423 : Bool;
      b1424 : Bool;
      b1425 : Bool;
      b1426 : Bool;
      b1427 : Bool;
      b1430 : Bool;
      b1431 : Bool;
      b1432 : Bool;
      b1433 : Bool;
      b1434 : Bool;
      b1435 : Bool;
      b1436 : Bool;
      b1437 : Bool;
      b1440 : Bool;
      b1441 : Bool;
      b1442 : Bool;
      b1443 : Bool;
      b1444 : Bool;
      b1445 : Bool;
      b1446 : Bool;
      b1447 : Bool;
      b1450 : Bool;
      b1451 : Bool;
      b1452 : Bool;
      b1453 : Bool;
      b1454 : Bool;
      b1455 : Bool;
      b1456 : Bool;
      b1457 : Bool;
      b1460 : Bool;
      b1461 : Bool;
      b1462 : Bool;
      b1463 : Bool;
      b1464 : Bool;
      b1465 : Bool;
      b1466 : Bool;
      b1467 : Bool;
      b1470 : Bool;
      b1471 : Bool;
      b1472 : Bool;
      b1473 : Bool;
      b1474 : Bool;
      b1475 : Bool;
      b1476 : Bool;
      b1477 : Bool;
      b1480 : Bool;
      b1481 : Bool;
      b1482 : Bool;
      b1483 : Bool;
      b1484 : Bool;
      b1485 : Bool;
      b1486 : Bool;
      b1487 : Bool;
      b1490 : Bool;
      b1491 : Bool;
      b1492 : Bool;
      b1493 : Bool;
      b1494 : Bool;
      b1495 : Bool;
      b1496 : Bool;
      b1497 : Bool;
      M338 : Bool;
      b1501 : Bool;
      b1502 : Bool;
      b1503 : Bool;
      b1504 : Bool;
      b1505 : Bool;
      b1506 : Bool;
      b1507 : Bool;
      b1510 : Bool;
      b1511 : Bool;
      b1512 : Bool;
      b1513 : Bool;
      b1514 : Bool;
      b1515 : Bool;
      b1516 : Bool;
      b1517 : Bool;
      b1520 : Bool;
      b1521 : Bool;
      b1522 : Bool;
      b1523 : Bool;
      b1524 : Bool;
      b1525 : Bool;
      b1526 : Bool;
      b1527 : Bool;
      b1530 : Bool;
      b1531 : Bool;
      b1532 : Bool;
      b1533 : Bool;
      b1534 : Bool;
      b1535 : Bool;
      b1536 : Bool;
      b1537 : Bool;
      b1540 : Bool;
      b1541 : Bool;
      b1542 : Bool;
      b1543 : Bool;
      b1544 : Bool;
      b1545 : Bool;
      b1546 : Bool;
      b1547 : Bool;
      b1550 : Bool;
      b1551 : Bool;
      b1552 : Bool;
      b1553 : Bool;
      b1554 : Bool;
      b1555 : Bool;
      b1556 : Bool;
      b1557 : Bool;
      b1560 : Bool;
      b1561 : Bool;
      b1562 : Bool;
      b1563 : Bool;
      b1564 : Bool;
      b1565 : Bool;
      b1566 : Bool;
      b1567 : Bool;
      b1570 : Bool;
      b1571 : Bool;
      b1572 : Bool;
      b1573 : Bool;
      b1574 : Bool;
      b1575 : Bool;
      b1576 : Bool;
      b1577 : Bool;
      b1580 : Bool;
      b1581 : Bool;
      b1582 : Bool;
      b1583 : Bool;
      b1584 : Bool;
      b1585 : Bool;
      b1586 : Bool;
      b1587 : Bool;
      b1590 : Bool;
      b1591 : Bool;
      b1592 : Bool;
      b1593 : Bool;
      b1594 : Bool;
      b1595 : Bool;
      b1596 : Bool;
      b1597 : Bool;
      b1600 : Bool;
      b1601 : Bool;
      b1602 : Bool;
      b1603 : Bool;
      b1604 : Bool;
      b1605 : Bool;
      b1606 : Bool;
      b1607 : Bool;
      b1610 : Bool;
      b1611 : Bool;
      b1612 : Bool;
      b1613 : Bool;
      b1614 : Bool;
      b1615 : Bool;
      b1616 : Bool;
      b1617 : Bool;
      b1620 : Bool;
      b1621 : Bool;
      b1622 : Bool;
      b1623 : Bool;
      b1624 : Bool;
      b1625 : Bool;
      b1626 : Bool;
      b1627 : Bool;
      b1630 : Bool;
      b1631 : Bool;
      b1632 : Bool;
      b1633 : Bool;
      b1634 : Bool;
      b1635 : Bool;
      b1636 : Bool;
      b1637 : Bool;
      b1640 : Bool;
      b1641 : Bool;
      b1642 : Bool;
      b1643 : Bool;
      b1644 : Bool;
      b1645 : Bool;
      b1646 : Bool;
      b1647 : Bool;
      b1650 : Bool;
      b1651 : Bool;
      b1652 : Bool;
      b1653 : Bool;
      b1654 : Bool;
      b1655 : Bool;
      b1656 : Bool;
      b1657 : Bool;
      b1660 : Bool;
      b1661 : Bool;
      b1662 : Bool;
      b1663 : Bool;
      b1664 : Bool;
      b1665 : Bool;
      b1666 : Bool;
      b1667 : Bool;
      b1670 : Bool;
      b1671 : Bool;
      b1672 : Bool;
      b1673 : Bool;
      b1674 : Bool;
      b1675 : Bool;
      b1676 : Bool;
      b1677 : Bool;
      b1680 : Bool;
      b1681 : Bool;
      b1682 : Bool;
      b1683 : Bool;
      b1684 : Bool;
      b1685 : Bool;
      b1686 : Bool;
      b1687 : Bool;
      b1690 : Bool;
      b1691 : Bool;
      b1692 : Bool;
      b1693 : Bool;
      b1694 : Bool;
      b1695 : Bool;
      b1696 : Bool;
      b1697 : Bool;
      b1700 : Bool;
      b1701 : Bool;
      b1702 : Bool;
      b1703 : Bool;
      b1704 : Bool;
      b1705 : Bool;
      b1706 : Bool;
      b1707 : Bool;
      b1710 : Bool;
      b1711 : Bool;
      b1712 : Bool;
      b1713 : Bool;
      b1714 : Bool;
      b1715 : Bool;
      b1716 : Bool;
      b1717 : Bool;
      b1720 : Bool;
      b1721 : Bool;
      b1722 : Bool;
      b1723 : Bool;
      b1724 : Bool;
      b1725 : Bool;
      b1726 : Bool;
      b1727 : Bool;
      b1730 : Bool;
      b1731 : Bool;
      b1732 : Bool;
      b1733 : Bool;
      b1734 : Bool;
      b1735 : Bool;
      b1736 : Bool;
      b1737 : Bool;
      b1740 : Bool;
      b1741 : Bool;
      b1742 : Bool;
      b1743 : Bool;
      b1744 : Bool;
      b1745 : Bool;
      b1746 : Bool;
      b1747 : Bool;
      b1750 : Bool;
      b1751 : Bool;
      b1752 : Bool;
      b1753 : Bool;
      b1754 : Bool;
      b1755 : Bool;
      b1756 : Bool;
      b1757 : Bool;
      b1760 : Bool;
      b1761 : Bool;
      b1762 : Bool;
      b1763 : Bool;
      b1764 : Bool;
      b1765 : Bool;
      b1766 : Bool;
      b1767 : Bool;
      b1770 : Bool;
      b1771 : Bool;
      b1772 : Bool;
      b1773 : Bool;
      b1774 : Bool;
      b1775 : Bool;
      b1776 : Bool;
      b1777 : Bool;
      b1780 : Bool;
      b1781 : Bool;
      b1782 : Bool;
      b1783 : Bool;
      b1784 : Bool;
      b1785 : Bool;
      b1786 : Bool;
      b1787 : Bool;
      b1790 : Bool;
      b1791 : Bool;
      b1792 : Bool;
      b1793 : Bool;
      b1794 : Bool;
      b1795 : Bool;
      b1796 : Bool;
      b1797 : Bool;
      b1800 : Bool;
      b1801 : Bool;
      b1802 : Bool;
      b1803 : Bool;
      b1804 : Bool;
      b1805 : Bool;
      b1806 : Bool;
      b1807 : Bool;
      b1810 : Bool;
      b1811 : Bool;
      b1812 : Bool;
      b1813 : Bool;
      b1814 : Bool;
      b1815 : Bool;
      b1816 : Bool;
      b1817 : Bool;
      b1820 : Bool;
      b1821 : Bool;
      b1822 : Bool;
      b1823 : Bool;
      b1824 : Bool;
      b1825 : Bool;
      b1826 : Bool;
      b1827 : Bool;
      b1830 : Bool;
      b1831 : Bool;
      b1832 : Bool;
      b1833 : Bool;
      b1834 : Bool;
      b1835 : Bool;
      b1836 : Bool;
      b1837 : Bool;
      b1840 : Bool;
      b1841 : Bool;
      b1842 : Bool;
      b1843 : Bool;
      b1844 : Bool;
      b1845 : Bool;
      b1846 : Bool;
      b1847 : Bool;
      b1850 : Bool;
      b1851 : Bool;
      b1852 : Bool;
      b1853 : Bool;
      b1854 : Bool;
      b1855 : Bool;
      b1856 : Bool;
      b1857 : Bool;
      b1860 : Bool;
      b1861 : Bool;
      b1862 : Bool;
      b1863 : Bool;
      b1864 : Bool;
      b1865 : Bool;
      b1866 : Bool;
      b1867 : Bool;
      b1870 : Bool;
      b1871 : Bool;
      b1872 : Bool;
      b1873 : Bool;
      b1874 : Bool;
      b1875 : Bool;
      b1876 : Bool;
      b1877 : Bool;
      b1880 : Bool;
      b1881 : Bool;
      b1882 : Bool;
      b1883 : Bool;
      b1884 : Bool;
      b1885 : Bool;
      b1886 : Bool;
      b1887 : Bool;
      b1890 : Bool;
      b1891 : Bool;
      b1892 : Bool;
      b1893 : Bool;
      b1894 : Bool;
      b1895 : Bool;
      b1896 : Bool;
      b1897 : Bool;
   END_STRUCT;


BEGIN
   b00 := TRUE;
   b01 := TRUE;
   b02 := TRUE;
   b03 := TRUE;
   b11 := TRUE;
   b13 := TRUE;
   b22 := TRUE;
   b81 := TRUE;
   b82 := TRUE;
   b84 := TRUE;
   b104 := TRUE;
   b106 := TRUE;
   b110 := TRUE;
   b113 := TRUE;
   b124 := TRUE;
   b126 := TRUE;
   b127 := TRUE;
   b161 := TRUE;
   b165 := TRUE;
   b184 := TRUE;
   b185 := TRUE;
   b186 := TRUE;
   b190 := TRUE;
   b191 := TRUE;
   b192 := TRUE;
   b194 := TRUE;
   b202 := TRUE;
   b226 := TRUE;
   b231 := TRUE;
   b244 := TRUE;
   b245 := TRUE;
   b261 := TRUE;
   b310 := TRUE;
   b320 := TRUE;
   b322 := TRUE;
   b326 := TRUE;
   b425 := TRUE;
   b426 := TRUE;
   b427 := TRUE;
   b432 := TRUE;
   b433 := TRUE;
   b434 := TRUE;
   b435 := TRUE;
   b436 := TRUE;
   b437 := TRUE;
   b440 := TRUE;
   b460 := TRUE;
   b580 := TRUE;
   b720 := TRUE;
   b721 := TRUE;
   b727 := TRUE;
   b770 := TRUE;
   b772 := TRUE;
   b782 := TRUE;
   b783 := TRUE;
   b784 := TRUE;
   b785 := TRUE;
   b801 := TRUE;
   b1301 := TRUE;
   b1321 := TRUE;
   b1323 := TRUE;
   b1325 := TRUE;
   b1326 := TRUE;
   b1404 := TRUE;
   b1464 := TRUE;
   b1480 := TRUE;
   b1542 := TRUE;
   b1550 := TRUE;
   b1582 := TRUE;
   b1590 := TRUE;

END_DATA_BLOCK

